// TwinCAT 3 PLC project PLC
// ProgramVersion: 3.1.4026.19
// libraries:
//   Tc2_Standard, * (Beckhoff Automation GmbH)
//   Tc2_System, * (Beckhoff Automation GmbH)
// project tree:
//   / PlcTask.TcTTO
//   POUs/ MAIN.TcPOU, SecondPouCreatedFromUser1.TcPOU
// real-time tasks:
//   TASK PlcTask: cycle T#10ms, priority 20, ADS port 350

CONFIGURATION PLC
    RESOURCE PLC ON TwinCAT3
        TASK PlcTask(INTERVAL := T#10ms, PRIORITY := 20);
        PROGRAM MAIN WITH PlcTask : MAIN;
    END_RESOURCE
END_CONFIGURATION

// ---- POUs/MAIN.TcPOU
PROGRAM MAIN
VAR
	CounterFromUser1	: DINT;
	newvarlocaltarget	: LREAL;
	newvar	: DINT;
	newvarFromUser1: DINT;
END_VAR

CounterFromUser1	:= CounterFromUser1 +2;

END_PROGRAM

// ---- POUs/SecondPouCreatedFromUser1.TcPOU
PROGRAM SecondPouCreatedFromUser1
VAR
END_VAR

END_PROGRAM
